{attribute 'qualified_only'}
{attribute 'strict'}
TYPE Cmd :
(
	None,
	Abort,
	Reset,
	Start,
	Stop,
	Pause,
	Resume
);
END_TYPE

(* stored: Version 1.1.0.1, ProductVersion 3.1.4022.11
   DUT Cmd: Id {1e5b96b8-90c8-4326-8491-d48b6b264de9} *)
